TYPE (* DataPanel Modules with medium IO density DI Struct + Source Address *)
  (* Version 1.0, 2026-05-28, franz *)
  PACKAGE DataPanel::io::MI::DI;
  IMPORT DataPanel::io::MI::DI::DataPanel_MI_DI::Invalid;
  IMPORT DataPanel::io::MI::const::MI::MI_00;
  IMPORT eclipse4diac::core::TypeHash;
  DataPanel_MI_DI_S_Octal_SA : STRUCT
    u8SAMember : USINT := MI_00; (* Node SA 224..239 *)
    Port1 : DataPanel::io::MI::DI::DataPanel_MI_DI_S := Invalid; (* Identify the Port 1A..8B *)
    Port2 : DataPanel::io::MI::DI::DataPanel_MI_DI_S := Invalid; (* Identify the Port 1A..8B *)
    Port3 : DataPanel::io::MI::DI::DataPanel_MI_DI_S := Invalid; (* Identify the Port 1A..8B *)
    Port4 : DataPanel::io::MI::DI::DataPanel_MI_DI_S := Invalid; (* Identify the Port 1A..8B *)
    Port5 : DataPanel::io::MI::DI::DataPanel_MI_DI_S := Invalid; (* Identify the Port 1A..8B *)
    Port6 : DataPanel::io::MI::DI::DataPanel_MI_DI_S := Invalid; (* Identify the Port 1A..8B *)
    Port7 : DataPanel::io::MI::DI::DataPanel_MI_DI_S := Invalid; (* Identify the Port 1A..8B *)
    Port8 : DataPanel::io::MI::DI::DataPanel_MI_DI_S := Invalid; (* Identify the Port 1A..8B *)
  END_STRUCT;
END_TYPE
